// TIA Portal V19 export
DATA_BLOCK "TIMER_MIN_DB_1"   // DB42
// stored: InstanceOfName TIMER_MIN, InstanceOfType FB
"TIMER_MIN"
   // VAR_INPUT
   //    "SET TIME" : Int;
   //    RESET : Bool;
   //    INPUT : Bool;
   // END_VAR
   // VAR_OUTPUT
   //    "PRESENT VALUE OF TIME" : Int;
   //    DONE : Bool;
   // END_VAR
   // VAR RETAIN
   //    "TIMER" { S7_SetPoint := 'True'} : IEC_TIMER;
   //    COUNTER1 { S7_SetPoint := 'True'} : IEC_COUNTER;
   // END_VAR
BEGIN
END_DATA_BLOCK
